(* Schneider Machine Expert - Basic project level_control, file version 2.9.0.0 *)
(* ProjectInformations: Name=Novo projeto *)

HARDWARE
  Cpu 0: TM221M16R/G
  ModuleExtensionObject 0: TM3DI8/G
  EthernetConfiguration: NetworkName=M221, IpAllocationMode=FixedAddress, IpAddress=0.0.0.0, SubnetMask=0.0.0.0
  SerialLineConfiguration: Baud=Baud19200, Parity=ParityEven, DataBits=DataBits8, StopBits=StopBits1, PhysicalMedium=PhysicalMediumRs485, TransmissionMode=TransmissionModeModbusRtu, SlaveId=1, Addressing=SlaveAddressing
  MastTask: UsePeriodScanMode=false, PeriodScan=100
  FastTask: Period=255
  CpuBehavior: StartingMode=StartAsPreviousState, AutoSaveRamOnEeprom=true, WatchdogPeriod=250

SYMBOLS  (address, symbol, comment, settings)
  %M0       INPUT_SENS_S1_TQ_PRINC  "Sensor de leitura de nível em 80%"
  %M1       INPUT_SENS_S2_TQ1_PRINC  "Sensor de leitura de nível em 50%"
  %M2       INPUT_SENS_S3_TQ1_PRINC  "Sensor de leitura de nível em 20%"
  %M3       INPUT_SENS_SH_TQ_COAG1
  %M4       INPUT_SENS_SL_TQ_COAG1
  %M5       INPUT_SENS_SH_TQ_COAG2
  %M6       INPUT_SENS_SL_TQ_COAG2
  %M7       INPUT_SENS_SH_TQ_POLI1
  %M8       INPUT_SENS_SL_TQ_POLI1
  %M9       INPUT_SENS_SH_TQ_POLI2
  %M10      INPUT_SENS_SL_TQ_POLI2
  %M11      INPUT_SENS_SL_TQ_TERC  "Sensor de Leitura de nível em 20%"

POU Entradas
  (* SectionNumber=0 *)

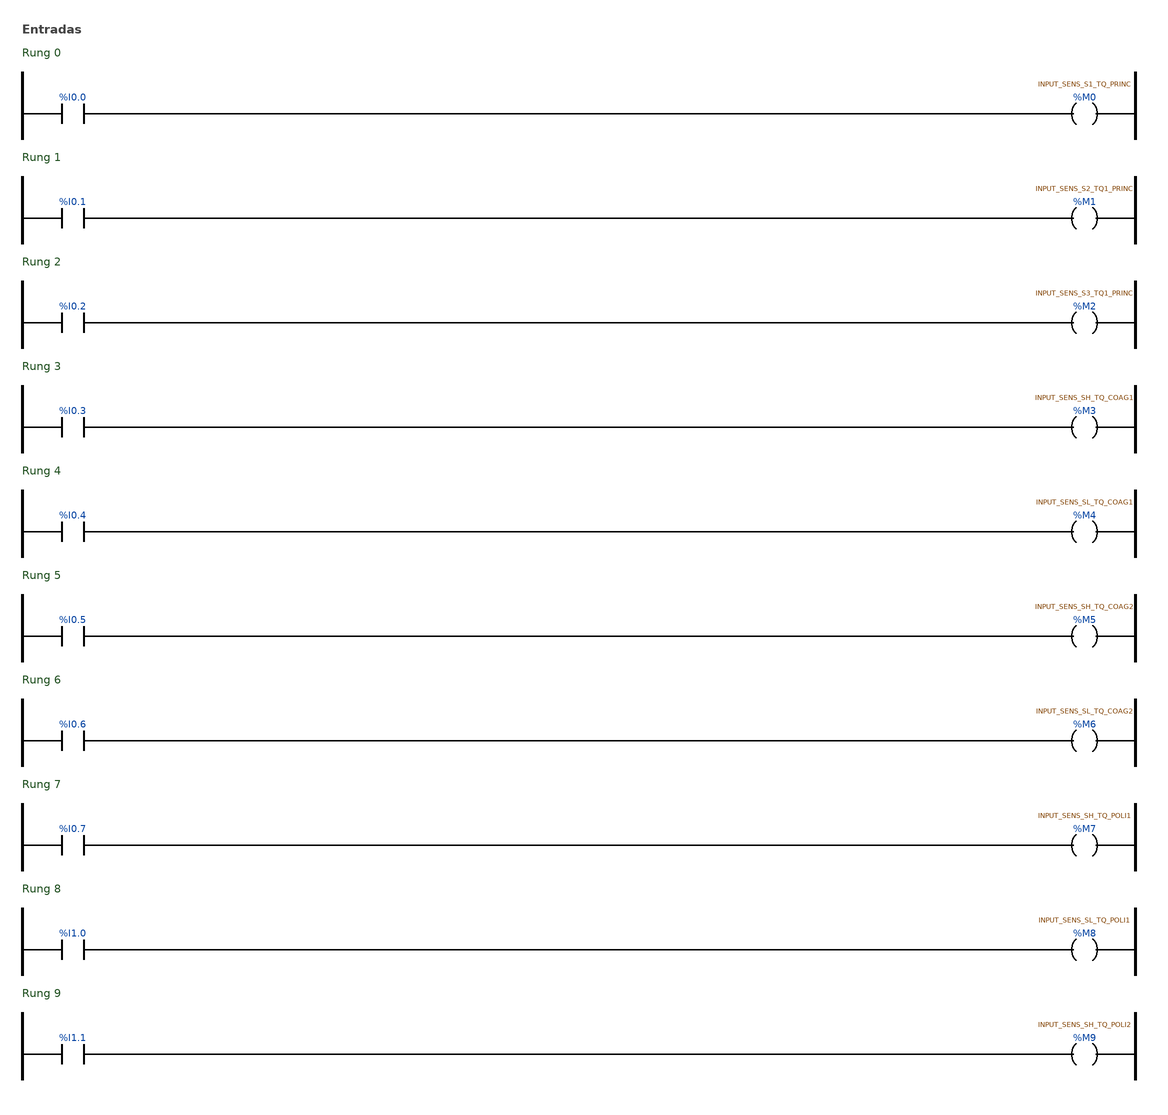

// Rung 0
  LD %I0.0
  ST %M0                  (* INPUT_SENS_S1_TQ_PRINC *)
  // as ST:
  //   INPUT_SENS_S1_TQ_PRINC := %I0.0;

// Rung 1
  LD %I0.1
  ST %M1                  (* INPUT_SENS_S2_TQ1_PRINC *)
  // as ST:
  //   INPUT_SENS_S2_TQ1_PRINC := %I0.1;

// Rung 2
  LD %I0.2
  ST %M2                  (* INPUT_SENS_S3_TQ1_PRINC *)
  // as ST:
  //   INPUT_SENS_S3_TQ1_PRINC := %I0.2;

// Rung 3
  LD %I0.3
  ST %M3                  (* INPUT_SENS_SH_TQ_COAG1 *)
  // as ST:
  //   INPUT_SENS_SH_TQ_COAG1 := %I0.3;

// Rung 4
  LD %I0.4
  ST %M4                  (* INPUT_SENS_SL_TQ_COAG1 *)
  // as ST:
  //   INPUT_SENS_SL_TQ_COAG1 := %I0.4;

// Rung 5
  LD %I0.5
  ST %M5                  (* INPUT_SENS_SH_TQ_COAG2 *)
  // as ST:
  //   INPUT_SENS_SH_TQ_COAG2 := %I0.5;

// Rung 6
  LD %I0.6
  ST %M6                  (* INPUT_SENS_SL_TQ_COAG2 *)
  // as ST:
  //   INPUT_SENS_SL_TQ_COAG2 := %I0.6;

// Rung 7
  LD %I0.7
  ST %M7                  (* INPUT_SENS_SH_TQ_POLI1 *)
  // as ST:
  //   INPUT_SENS_SH_TQ_POLI1 := %I0.7;

// Rung 8
  LD %I1.0
  ST %M8                  (* INPUT_SENS_SL_TQ_POLI1 *)
  // as ST:
  //   INPUT_SENS_SL_TQ_POLI1 := %I1.0;

// Rung 9
  LD %I1.1
  ST %M9                  (* INPUT_SENS_SH_TQ_POLI2 *)
  // as ST:
  //   INPUT_SENS_SH_TQ_POLI2 := %I1.1;

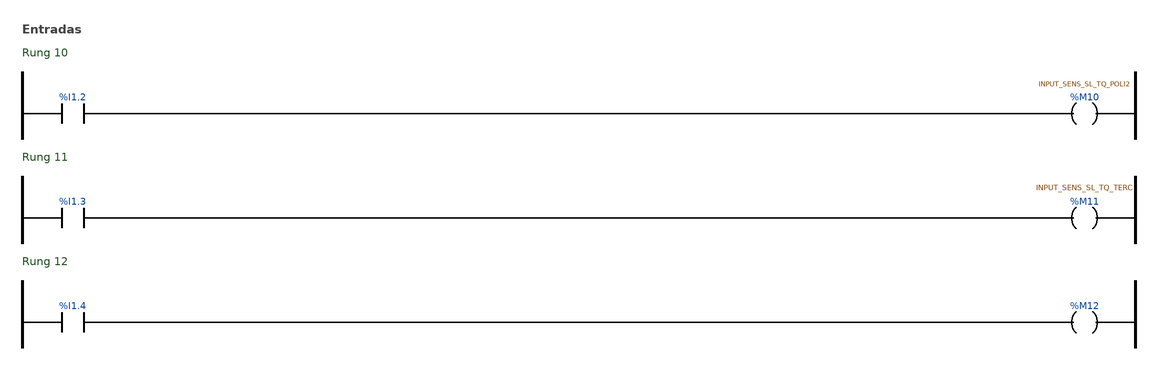

// Rung 10
  LD %I1.2
  ST %M10                 (* INPUT_SENS_SL_TQ_POLI2 *)
  // as ST:
  //   INPUT_SENS_SL_TQ_POLI2 := %I1.2;

// Rung 11
  LD %I1.3
  ST %M11                 (* INPUT_SENS_SL_TQ_TERC *)
  // as ST:
  //   INPUT_SENS_SL_TQ_TERC := %I1.3;

// Rung 12
  LD %I1.4
  ST %M12
  // as ST:
  //   %M12 := %I1.4;

POU Lógica
  (* SectionNumber=0 *)

// Rung 13
  LD

POU Saídas
  (* SectionNumber=0 *)

// Rung 14
  LD
